SUBAPPLICATION SlurryTanker (* Subapplication Type *)
  (* Standard: 61499-2 *)
  (* Version 1.0, 2023-02-11, franz *)
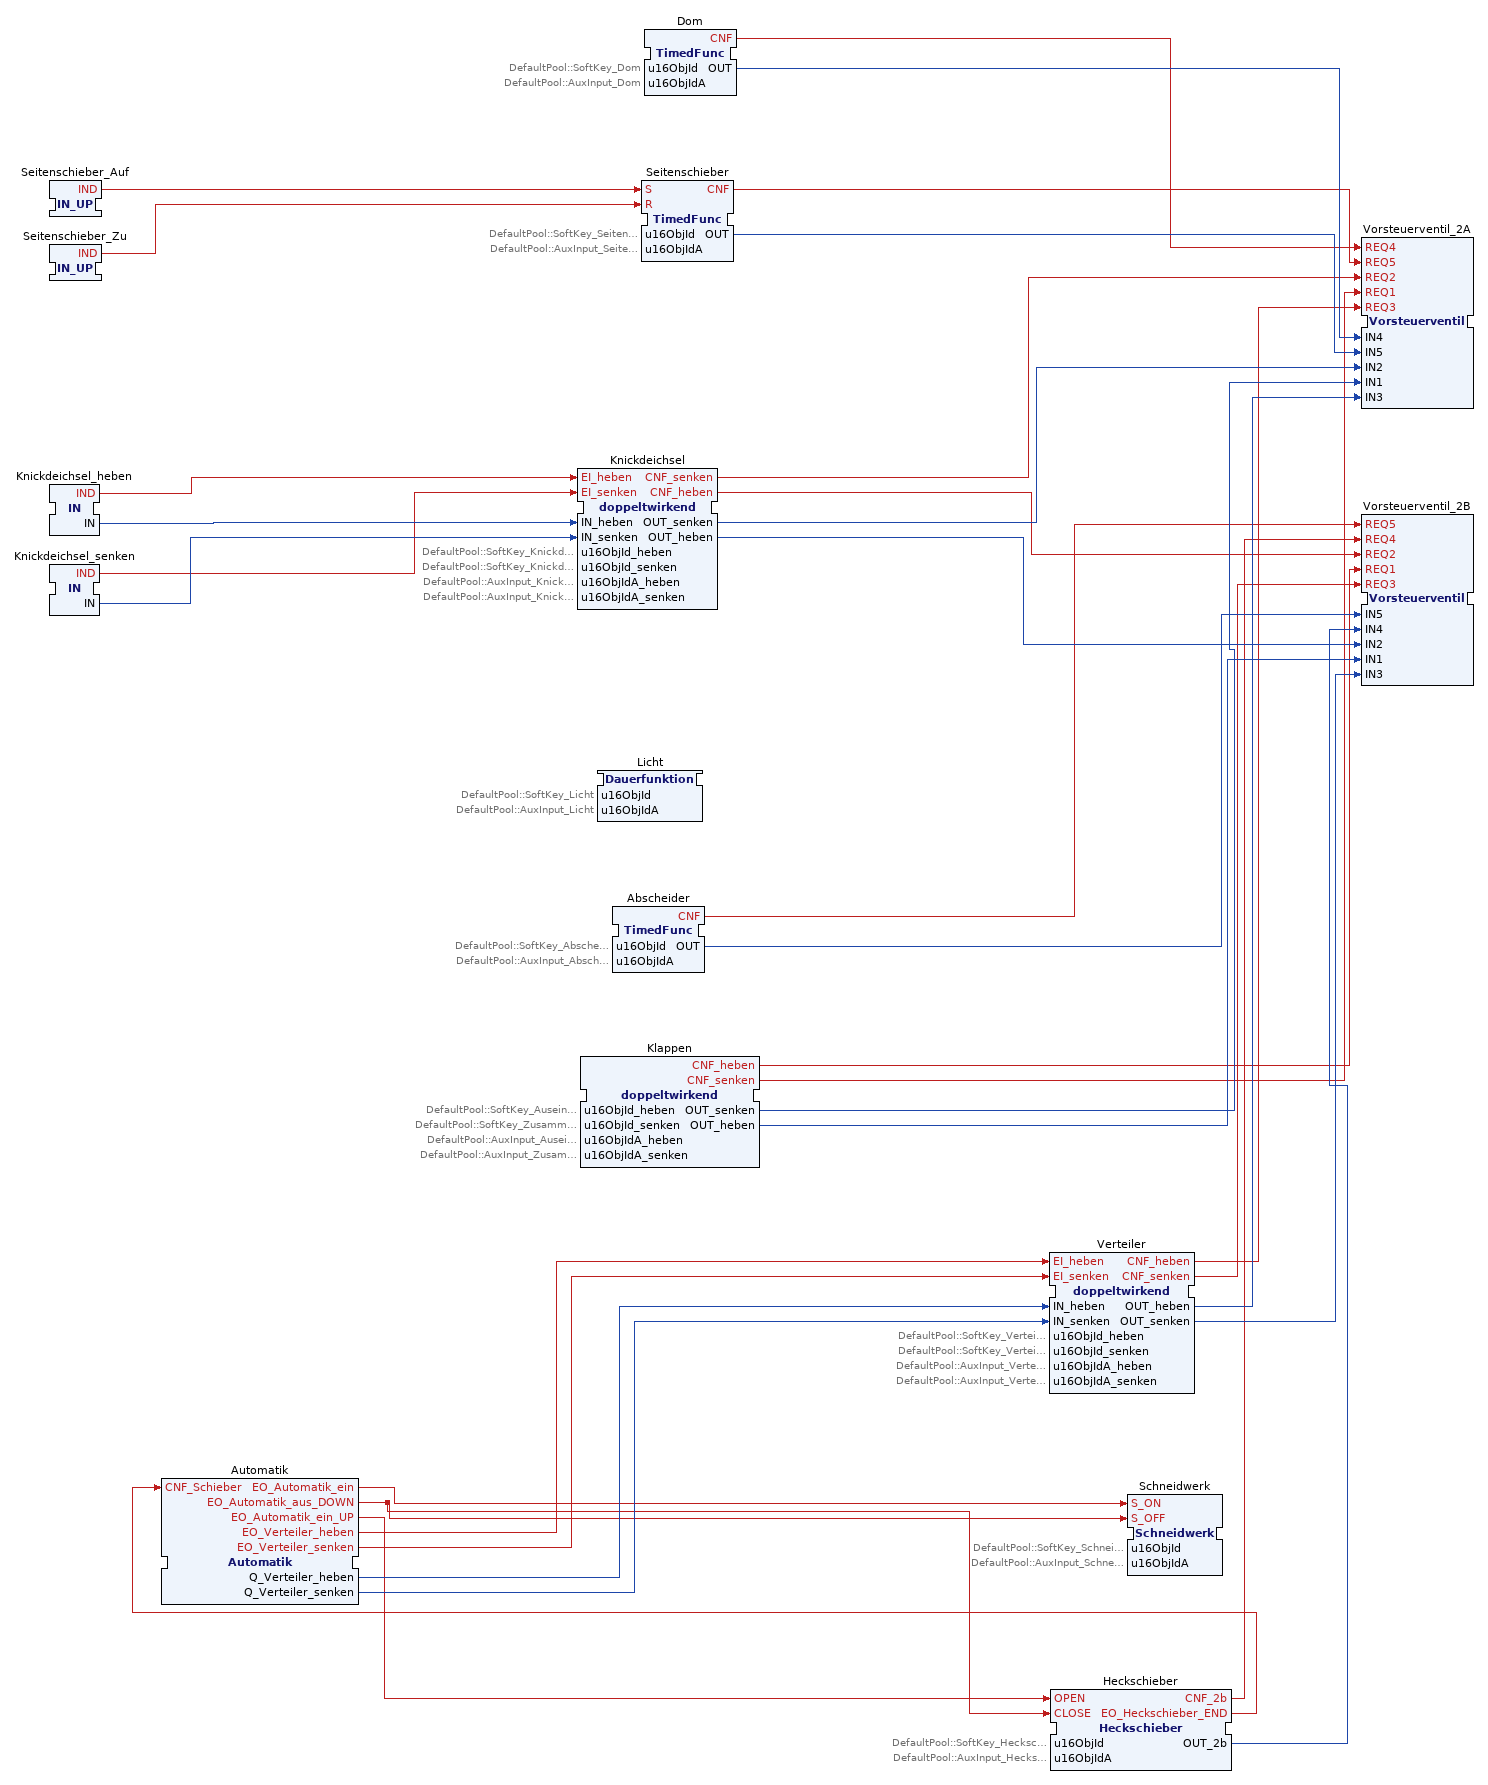
  (* Group funktionen: *)
  (* Group Vorsteuerventile: Vorsteuerventile *)
  (* Group Vorgewendeautomatik: Vorgewendeautomatik *)
  SUBAPPS
    Automatik : Automatik; {SET_ATTRIBUTE(GroupName, Vorgewendeautomatik)}
    Dom : TimedFunc(u16ObjId := DefaultPool::SoftKey_Dom, u16ObjIdA := DefaultPool::AuxInput_Dom); {SET_ATTRIBUTE(GroupName, funktionen)}
    Seitenschieber : TimedFunc(u16ObjId := DefaultPool::SoftKey_Seitenschieber, u16ObjIdA := DefaultPool::AuxInput_Seitenschieber); {SET_ATTRIBUTE(GroupName, funktionen)}
    Klappen : doppeltwirkend(u16ObjId_heben := DefaultPool::SoftKey_Auseinanderklappen, u16ObjId_senken := DefaultPool::SoftKey_Zusammenklappen, u16ObjIdA_heben := DefaultPool::AuxInput_Auseinanderklappen, u16ObjIdA_senken := DefaultPool::AuxInput_Zusammenklappen); {SET_ATTRIBUTE(GroupName, funktionen)}
    Verteiler : doppeltwirkend(u16ObjId_heben := DefaultPool::SoftKey_Verteiler_heben, u16ObjId_senken := DefaultPool::SoftKey_Verteiler_senken, u16ObjIdA_heben := DefaultPool::AuxInput_Verteiler_heben, u16ObjIdA_senken := DefaultPool::AuxInput_Verteiler_senken); {SET_ATTRIBUTE(GroupName, Vorgewendeautomatik)}
    Vorsteuerventil_2A : Vorsteuerventil; {SET_ATTRIBUTE(GroupName, Vorsteuerventile)}
    Vorsteuerventil_2B : Vorsteuerventil; {SET_ATTRIBUTE(GroupName, Vorsteuerventile)}
    Knickdeichsel : doppeltwirkend(u16ObjId_heben := DefaultPool::SoftKey_Knickdeichsel_heben, u16ObjId_senken := DefaultPool::SoftKey_Knickdeichsel_senken, u16ObjIdA_heben := DefaultPool::AuxInput_Knickdeichsel_heben, u16ObjIdA_senken := DefaultPool::AuxInput_Knickdeichsel_senken); {SET_ATTRIBUTE(GroupName, funktionen)}
    Licht : Dauerfunktion(u16ObjId := DefaultPool::SoftKey_Licht, u16ObjIdA := DefaultPool::AuxInput_Licht); {SET_ATTRIBUTE(GroupName, funktionen)}
    Abscheider : TimedFunc(u16ObjId := DefaultPool::SoftKey_Abscheider, u16ObjIdA := DefaultPool::AuxInput_Abscheider); {SET_ATTRIBUTE(GroupName, funktionen)}
    Schneidwerk : Schneidwerk(u16ObjId := DefaultPool::SoftKey_Schneidwerk, u16ObjIdA := DefaultPool::AuxInput_Schneidwerk); {SET_ATTRIBUTE(GroupName, Vorgewendeautomatik)}
    Heckschieber : Heckschieber(u16ObjId := DefaultPool::SoftKey_Heckschieber, u16ObjIdA := DefaultPool::AuxInput_Heckschieber); {SET_ATTRIBUTE(GroupName, Vorgewendeautomatik)}
    Knickdeichsel_heben : IN; {SET_ATTRIBUTE(GroupName, funktionen)}
    Knickdeichsel_senken : IN; {SET_ATTRIBUTE(GroupName, funktionen)}
    Seitenschieber_Auf : IN_UP; {SET_ATTRIBUTE(GroupName, funktionen)}
    Seitenschieber_Zu : IN_UP; {SET_ATTRIBUTE(GroupName, funktionen)}
  END_SUBAPPS
  EVENT_CONNECTIONS
    Dom.CNF TO Vorsteuerventil_2A.REQ4;
    Seitenschieber.CNF TO Vorsteuerventil_2A.REQ5;
    Abscheider.CNF TO Vorsteuerventil_2B.REQ5;
    Automatik.EO_Automatik_ein TO Schneidwerk.S_ON;
    Automatik.EO_Automatik_aus_DOWN TO Schneidwerk.S_OFF;
    Automatik.EO_Automatik_ein_UP TO Heckschieber.OPEN;
    Automatik.EO_Automatik_aus_DOWN TO Heckschieber.CLOSE;
    Heckschieber.CNF_2b TO Vorsteuerventil_2B.REQ4;
    Heckschieber.EO_Heckschieber_END TO Automatik.CNF_Schieber;
    Automatik.EO_Verteiler_heben TO Verteiler.EI_heben;
    Automatik.EO_Verteiler_senken TO Verteiler.EI_senken;
    Knickdeichsel_heben.IND TO Knickdeichsel.EI_heben;
    Knickdeichsel_senken.IND TO Knickdeichsel.EI_senken;
    Knickdeichsel.CNF_senken TO Vorsteuerventil_2A.REQ2;
    Knickdeichsel.CNF_heben TO Vorsteuerventil_2B.REQ2;
    Klappen.CNF_heben TO Vorsteuerventil_2B.REQ1;
    Klappen.CNF_senken TO Vorsteuerventil_2A.REQ1;
    Verteiler.CNF_heben TO Vorsteuerventil_2A.REQ3;
    Verteiler.CNF_senken TO Vorsteuerventil_2B.REQ3;
    Seitenschieber_Auf.IND TO Seitenschieber.S;
    Seitenschieber_Zu.IND TO Seitenschieber.R;
  END_CONNECTIONS
  DATA_CONNECTIONS
    Dom.OUT TO Vorsteuerventil_2A.IN4;
    Seitenschieber.OUT TO Vorsteuerventil_2A.IN5;
    Abscheider.OUT TO Vorsteuerventil_2B.IN5;
    Heckschieber.OUT_2b TO Vorsteuerventil_2B.IN4;
    Automatik.Q_Verteiler_heben TO Verteiler.IN_heben;
    Automatik.Q_Verteiler_senken TO Verteiler.IN_senken;
    Knickdeichsel_heben.IN TO Knickdeichsel.IN_heben;
    Knickdeichsel_senken.IN TO Knickdeichsel.IN_senken;
    Knickdeichsel.OUT_senken TO Vorsteuerventil_2A.IN2;
    Knickdeichsel.OUT_heben TO Vorsteuerventil_2B.IN2;
    Klappen.OUT_senken TO Vorsteuerventil_2A.IN1;
    Klappen.OUT_heben TO Vorsteuerventil_2B.IN1;
    Verteiler.OUT_heben TO Vorsteuerventil_2A.IN3;
    Verteiler.OUT_senken TO Vorsteuerventil_2B.IN3;
  END_CONNECTIONS
END_SUBAPPLICATION
